FUNCTION_BLOCK Test_F_AssertAny_INTS_Differ EXTENDS T_UnitTestBase

METHOD Init
END_METHOD

METHOD RunTest
VAR_OUTPUT
    TestCompleted : BOOL;
    TestFailed    : BOOL;
END_VAR
VAR
    TestValue : INT;
    Actual    : INT;
END_VAR
TestValue := 133;
Actual    := 133;

AssertEquals(Source   := THIS^.TestName,
             Expected := TestValue,
             Actual   := Actual,
             Message  := 'Unexpected value of TestValue',
             Failed   => TestFailed);

TestCompleted := TRUE;
END_METHOD

END_FUNCTION_BLOCK

(* stored: Version 1.1.0.1, ProductVersion 3.1.4024.12
   POU Test_F_AssertAny_INTS_Differ: Id {84efddba-5fae-41db-9255-bfe641290d43}, SpecialFunc None
   Method Init: Id {0906e0bf-21d0-4331-9bda-44033c058ec6}
   Method RunTest: Id {5201941c-166a-4ae6-a43b-c98fa8f93239} *)
